{attribute 'Tc2GvlVarNames'}
VAR_GLOBAL
END_VAR

(* stored: Version 1.1.0.1, ProductVersion 3.1.4020.12
   GVL Globale_Variablen: Id {bea2aa21-1bff-4d6b-a26f-bd4f486da3f2} *)
